FUNCTION_BLOCK PUBLIC FINAL POU
VAR_INPUT
END_VAR
VAR_OUTPUT
END_VAR
VAR
END_VAR

END_FUNCTION_BLOCK

(* stored: Version 1.1.0.1, ProductVersion 3.1.4024.12
   POU POU: Id {5ad31d52-1a79-4fd6-a597-9b201947aeb1}, SpecialFunc None *)
